{region '#Template'}
	{attribute 'Category' := 'Universal'}
	{attribute 'Version' := '0.0.1.0'}
	{attribute 'Tags' := 'Universal, Sensor, BI, BV'}
	{attribute 'Description' := 'Kombination aus BV BI	// Combination of BV BI'}
{endregion}
FUNCTION_BLOCK FB_BA_CombinationBI_BV EXTENDS FB_BA_View
VAR_INPUT
END_VAR
VAR_INPUT CONSTANT
	Input				: FB_BA_BI_IO;	
	Value				: FB_BA_BV_Op;									
END_VAR
VAR_OUTPUT
	bBI_PrVal			: BOOL;
	bBV_PrVal			: BOOL;	
END_VAR
VAR
END_VAR

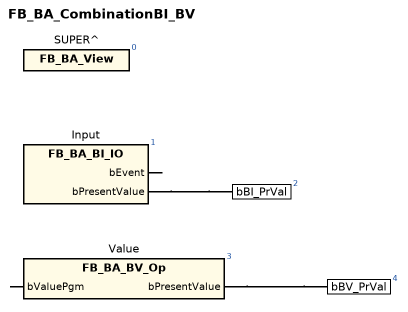
SUPER^(); // FB_BA_View
Input(); // FB_BA_BI_IO
bBI_PrVal := Input.bPresentValue;
Value(); // FB_BA_BV_Op
bBV_PrVal := Value.bPresentValue;

METHOD FB_init : BOOL
VAR_INPUT
	bInitRetains : BOOL; // if TRUE, the retain variables are initialized (warm start / cold start)
	bInCopyCode : BOOL;  // if TRUE, the instance afterwards gets moved into the copy code (online change)
END_VAR
Input.iParent						:= THIS^;
Input.iLabel						:= LblFunctions.Button;	
Input.sObjectName					:= '{Idx=01}';
Input.sDeviceType					:= '';	
Input.bEnOutOfService				:= FALSE;
Input.ePolarity						:= E_BA_Polarity.eReverse;
Input.sActiveText 					:= Texts.txtOn;
Input.sInactiveText 				:= Texts.txtOff;
Input.nStateChangeCount				:= 0;
Input.nActiveTimeElapsed			:= 0;
Input.nEventClassID					:= EventClasses.NotificationSimple;
Input.stTimeDelay.nToNormal			:= BA2_Param.nDefTimeDelay_ToNormal;
Input.stTimeDelay.nToAbnormal		:= BA2_Param.nDefTimeDelay_ToAbnormal;
Input.bAlarmValue					:= TRUE;
Input.bAcknowledgeRm				:= FALSE;		
Input.aEventTransitionText[1]		:= Texts.txtOff;
Input.aEventTransitionText[2]		:= Texts.txtNone;
Input.aEventTransitionText[3]		:= Texts.txtOn;
Input.bEventDetectionEnable			:= FALSE;
Input.eEnPlantLock					:= E_BA_LockPriority.eNoLock;	

Value.iParent						:= THIS^;		
Value.iLabel 						:= LblFunctions.Button;	
Value.sObjectName					:= '{Idx=02}';	
Value.sActiveText					:= Texts.txtOn;
Value.sInactiveText					:= Texts.txtOff;
Value.bValueRm						:= FALSE;
Value.eToggleMode 					:= E_BA_ToggleMode.eSwitch;
END_METHOD

END_FUNCTION_BLOCK

(* stored: Version 1.1.0.1, ProductVersion 3.1.4024.6
   POU FB_BA_CombinationBI_BV: Id {683640bc-82e8-4fb1-aad6-81e3fa03e3ba}, SpecialFunc None
   Method FB_init: Id {62af4ccf-a83f-474b-92f1-193c092f017d} *)
